// TIA Portal V20 export
TYPE "LWONIK_typeSafetySensor"
// stored: Access Published
   STRUCT
      anodeCvCoverBwd { ExternalWritable := 'False'} : Bool;
      cathodeCvCoverBwd { ExternalWritable := 'False'} : Bool;
      anodeCvCoverFwd { ExternalWritable := 'False'} : Bool;
      cathodeCvCoverFwd { ExternalWritable := 'False'} : Bool;
   END_STRUCT;
END_TYPE
